FUNCTION_BLOCK FB_Ambient
VAR_INPUT
END_VAR
VAR_OUTPUT
	{attribute 'OPC.UA.DA' := '1'}
	localState : ST_AmbientState;
END_VAR
VAR
	//sensors
	UpperRoomTemperature_SW : FB_TemperatureSensor; //south west
	LowerRoomTemperature_SW : FB_TemperatureSensor;
	UpperRoomTemperature_NW : FB_TemperatureSensor; //north west
	LowerRoomTemperature_NW : FB_TemperatureSensor;
	UpperRoomTemperature_NO : FB_TemperatureSensor;//north east
	LowerRoomTemperature_NO : FB_TemperatureSensor;
	UpperRoomTemperature_SO : FB_TemperatureSensor; //south east
	LowerRoomTemperature_SO : FB_TemperatureSensor;
	
	OutsideTemperature_North : FB_TemperatureSensor;
	OutsideTemperature_South : FB_TemperatureSensor;
	OutsideTemperature_West : FB_TemperatureSensor;
	
	InletAHUTemperature : AutomationBaseClasses.FB_TemperatureSensor; //inlet temperature from climate room internal AHU (Air Handling Unit)
	OutletAHUTemperature : AutomationBaseClasses.FB_TemperatureSensor; //outlet temperature from climate room internal AHU
	
	InletVentilationTemperature : AutomationBaseClasses.FB_TemperatureSensor; //inlet temperature from building ventilation
	OutletVentilationTemperature : AutomationBaseClasses.FB_TemperatureSensor; //outlet temperature from building ventilation
	
	RoomHumidity : FB_HumiditySensor;
	RoomCO2 : FB_CO2Sensor;
END_VAR

UpperRoomTemperature_SW();
UpperRoomTemperature_SW.GetState_AI();
LowerRoomTemperature_SW();
LowerRoomTemperature_SW.GetState_AI();
UpperRoomTemperature_NW();
UpperRoomTemperature_NW.GetState_AI();
LowerRoomTemperature_NW();
LowerRoomTemperature_NW.GetState_AI();
UpperRoomTemperature_NO();
UpperRoomTemperature_NO.GetState_AI();
LowerRoomTemperature_NO();
LowerRoomTemperature_NO.GetState_AI();
UpperRoomTemperature_SO();
UpperRoomTemperature_SO.GetState_AI();
LowerRoomTemperature_SO();
LowerRoomTemperature_SO.GetState_AI();

OutsideTemperature_North();
OutsideTemperature_North.GetState_AI();
OutsideTemperature_South();
OutsideTemperature_South.GetState_AI();
OutsideTemperature_West();
OutsideTemperature_West.GetState_AI();

InletAHUTemperature();
InletAHUTemperature.GetState_AI();
OutletAHUTemperature();
OutletAHUTemperature.GetState_AI();
InletVentilationTemperature();
InletVentilationTemperature.GetState_AI();
OutletVentilationTemperature();
OutletVentilationTemperature.GetState_AI();

RoomHumidity();
RoomHumidity.GetState_AI();

RoomCO2();
RoomCO2.GetState_AI();

SetState();

METHOD PROTECTED SetState : BOOL
VAR_INPUT
END_VAR
localState.fRelativeHumidity := RoomHumidity.fHumidity;
localState.fRoomCO2 := RoomCO2.fCO2;

localState.fRoomTemperatureUpperNO := UpperRoomTemperature_NO.fTemperature;
localState.fRoomTemperatureLowerNO := LowerRoomTemperature_NO.fTemperature;
localState.fRoomTemperatureUpperSO := UpperRoomTemperature_SO.fTemperature;
localState.fRoomTemperatureLowerSO := LowerRoomTemperature_SO.fTemperature;
localState.fRoomTemperatureUpperSW := UpperRoomTemperature_SW.fTemperature;
localState.fRoomTemperatureLowerSW := LowerRoomTemperature_SW.fTemperature;
localState.fRoomTemperatureUpperNW := UpperRoomTemperature_NW.fTemperature;
localState.fRoomTemperatureLowerNW := LowerRoomTemperature_NW.fTemperature;

localState.fInletAHUTemperature := InletAHUTemperature.fTemperature;
localState.fOutletAHUTemperature := OutletAHUTemperature.fTemperature;
localState.fInletVentilationTemperature := InletVentilationTemperature.fTemperature;
localState.fOutletVentilationTemperature := OutletVentilationTemperature.fTemperature;

//room temperature is currently calclated as mean value from all room values
localState.fRoomTemperature := (localState.fRoomTemperatureUpperNO+localState.fRoomTemperatureLowerNO+localState.fRoomTemperatureUpperSO+localState.fRoomTemperatureLowerSO+localState.fRoomTemperatureUpperSW+localState.fRoomTemperatureLowerSW+localState.fRoomTemperatureUpperNW+localState.fRoomTemperatureLowerNW)/8;

localState.fOutsideTemperatureNorth := OutsideTemperature_North.fTemperature;
localState.fOutsideTemperatureSouth := OutsideTemperature_South.fTemperature;
localState.fOutsideTemperatureWest := OutsideTemperature_West.fTemperature;

//outside temperature is currently calclated as mean value from all outside values
localState.fOutsideTemperature := (localState.fOutsideTemperatureNorth+localState.fOutsideTemperatureSouth+localState.fOutsideTemperatureWest)/3;
END_METHOD

END_FUNCTION_BLOCK

(* stored: Version 1.1.0.1, ProductVersion 3.1.4024.6
   POU FB_Ambient: Id {0f4d897f-37c6-49e7-b457-70281b1a7b2e}, SpecialFunc None
   Method SetState: Id {eda2988d-3dfb-4e58-a5fe-95deb2a32f09} *)
